// TIA Portal project "Soru2" (V15)

(* hardware
DEVICE "S7-1200 station_1"  S7-1200 Station
   slot 0: "Rack_0"  S7-1200 Rack  Rack  V1.0
   slot 1: "PLC_1"  CPU 1214C DC/DC/DC  6ES7 214-1AG40-0XB0  V4.2
*)

// ===== PLC "PLC_1"  CPU 1214C DC/DC/DC =====

VAR_GLOBAL   // PLC tag table "Default tag table"
   "Stop" AT %I0.0 : Bool;
   "Baslat" AT %I0.1 : Bool;
   "Motor_0" AT %Q0.0 : Bool;
   "Motor_1" AT %Q0.1 : Bool;
   "Motor_2" AT %Q0.2 : Bool;
   "Tag_1" AT %M0.0 : Bool;
   "1. Motor Calisiyor" AT %M0.1 : Bool;
   "Tag_3" AT %M0.2 : Bool;
   "2. Motor Calisiyor" AT %M0.3 : Bool;
   "3. Motor Calisiyor" AT %M0.4 : Bool;
END_VAR

ORGANIZATION_BLOCK "Main"   // OB1, LAD, ProgramCycle
TITLE = "Main Program Sweep (Cycle)"
{ S7_Optimized_Access := 'TRUE' }
VERSION : 0.1
   VAR_INPUT
      Initial_Call : Bool;   // Initial call of this OB
      Remanence : Bool;   // =True, if remanent data are available
   END_VAR
   VAR_TEMP   // added for the SCL form of the ladder/FBD networks
      _w1 : Bool;
      _w2 : Bool;
      _w3 : Bool;
   END_VAR
BEGIN

REGION Network 1
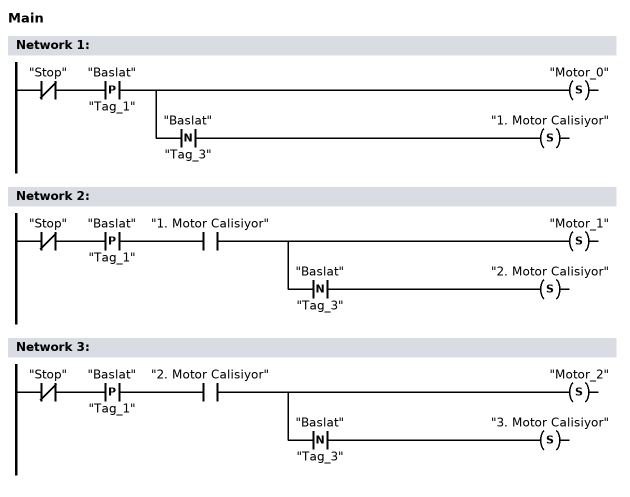
   RUNG wire#powerrail
      I_Contact( "Stop" )
      P_Contact(operand := "Baslat", bit := "Tag_1")
      wire#w1
      S_Coil( "Motor_0" )
   END_RUNG
   RUNG wire#w1
      N_Contact(operand := "Baslat", bit := "Tag_3")
      S_Coil( "1. Motor Calisiyor" )
   END_RUNG
   // the same network as SCL:
   #_w1 := NOT "Stop" AND "Baslat" AND NOT "Tag_1";   // rising edge of "Baslat"
   "Tag_1" := "Baslat";
   IF #_w1 THEN "Motor_0" := TRUE; END_IF;
   #_w2 := #_w1 AND NOT "Baslat" AND "Tag_3";   // falling edge of "Baslat"
   "Tag_3" := "Baslat";
   IF #_w2 THEN "1. Motor Calisiyor" := TRUE; END_IF;
END_REGION

REGION Network 2
   RUNG wire#powerrail
      I_Contact( "Stop" )
      P_Contact(operand := "Baslat", bit := "Tag_1")
      Contact( "1. Motor Calisiyor" )
      wire#w1
      S_Coil( "Motor_1" )
   END_RUNG
   RUNG wire#w1
      N_Contact(operand := "Baslat", bit := "Tag_3")
      S_Coil( "2. Motor Calisiyor" )
   END_RUNG
   // the same network as SCL:
   #_w1 := NOT "Stop" AND "Baslat" AND NOT "Tag_1";   // rising edge of "Baslat"
   "Tag_1" := "Baslat";
   #_w2 := #_w1 AND "1. Motor Calisiyor";
   IF #_w2 THEN "Motor_1" := TRUE; END_IF;
   #_w3 := #_w2 AND NOT "Baslat" AND "Tag_3";   // falling edge of "Baslat"
   "Tag_3" := "Baslat";
   IF #_w3 THEN "2. Motor Calisiyor" := TRUE; END_IF;
END_REGION

REGION Network 3
   RUNG wire#powerrail
      I_Contact( "Stop" )
      P_Contact(operand := "Baslat", bit := "Tag_1")
      Contact( "2. Motor Calisiyor" )
      wire#w1
      S_Coil( "Motor_2" )
   END_RUNG
   RUNG wire#w1
      N_Contact(operand := "Baslat", bit := "Tag_3")
      S_Coil( "3. Motor Calisiyor" )
   END_RUNG
   // the same network as SCL:
   #_w1 := NOT "Stop" AND "Baslat" AND NOT "Tag_1";   // rising edge of "Baslat"
   "Tag_1" := "Baslat";
   #_w2 := #_w1 AND "2. Motor Calisiyor";
   IF #_w2 THEN "Motor_2" := TRUE; END_IF;
   #_w3 := #_w2 AND NOT "Baslat" AND "Tag_3";   // falling edge of "Baslat"
   "Tag_3" := "Baslat";
   IF #_w3 THEN "3. Motor Calisiyor" := TRUE; END_IF;
END_REGION
END_ORGANIZATION_BLOCK